INTERFACE PUBLIC LogEventBuffer EXTENDS __SYSTEM.IQueryInterface

{attribute 'monitoring':='call'}
PROPERTY PUBLIC IsFull : BOOL
GET
END_GET
END_PROPERTY

METHOD PUBLIC Pop : LogEvent
END_METHOD

METHOD PUBLIC Push : BOOL
VAR_INPUT
	event : LogEvent;
END_VAR
END_METHOD

{attribute 'monitoring':='call'}
PROPERTY PUBLIC Size : UDINT
GET
END_GET
END_PROPERTY

END_INTERFACE

(* stored: Version 1.1.0.1
   Itf LogEventBuffer: Id {16066395-45f0-43f0-9757-aebb6b34a4d0}
   Property IsFull: Id {6e369abe-4e03-4827-9255-db6582bc65b0}
   Get Get: Id {1febb82c-2e49-4124-98f0-1cb8e5865cc3}
   Method Pop: Id {c19c601f-961f-4523-a3b4-b11196398b6b}
   Method Push: Id {d2c783af-60f5-40e1-a6be-94784b56196f}
   Property Size: Id {7716115a-9344-492f-941d-d79d37d865c2}
   Get Get: Id {060d0ed7-e3a9-498c-a01b-6fa649a60cf2} *)
